Staubli VAL3: prd_action.pgx

program prd_action(string x_sString (dimensions=1))
begin
  switch x_sString
    //启动生产
    case "启动生产"
      call production()
    break
    //暂停生产
    case "暂停生产"
      bPause=true
      stopMove()
      dioSet(io:doB_7_toolOn,0)
      if dioGet(io:doB_9_tableOn)==1
        dioSet(io:doB_9_tableOn,0)
      endIf
    break
    //停止生产
    case "停止生产"
      stopMove()
      dioSet(io:doB_7_toolOn,0)
      dioSet(io:doB_9_tableOn,0)
      bSuspend=false
      read:bCycle=false
      if taskStatus("txtLoad")!=-1
        taskKill("txtLoad")
        wait(taskStatus("txtLoad")==-1)
      endIf
      if taskStatus("motion")!=-1
        taskKill("motion")
        wait(taskStatus("motion")==-1)
      endIf
    break
    //急停处理
    case "急停处理"
      stopMove()
      if dioGet(io:doB_7_toolOn)==1
        dioSet(io:doB_7_toolOn,0)
      endIf
      if dioGet(io:doB_9_tableOn)==1
        dioSet(io:doB_9_tableOn,0)
      endIf
      bSuspend=true
      if bPause==true
        bPause=false
      endIf
      read:bCycle=false
      read:libSave()
      if taskStatus("txtLoad")!=-1
        taskKill("txtLoad")
        wait(taskStatus("txtLoad")==-1)
      endIf
      if taskStatus("motion")!=-1
        taskKill("motion")
        wait(taskStatus("motion")==-1)
      endIf
    break
  endSwitch
end
